Omron Sysmac Studio project Code (Sysmac)_1 (Sysmac Studio 1.64.0.64008, StandardProject)

# Controller new_Controller_0: NX1P2-9B24DT1 version 1.42
Task PrimaryTask (priority 4, period or condition 4000): Program0
Library OEN_Communication_V1_0_22 1.0.22 (contents left out)

TYPE ST_CNC_Cmd : STRUCT  (* CNC DATA *)
    Start : BOOL;  (* CNC Start *)
    Stop : BOOL;  (* CNC Stop *)
    Reset : BOOL;  (* CNC Reset *)
    Busy : BOOL;  (* CNC Busy *)
    FirstPhaseDone : BOOL;  (* CNC Done *)
    LastPhaseDone : BOOL;  (* CNC Done *)
    Progress : INT;  (* CNC Progress *)
    ErrorCode : INT;  (* Erros 1, Error2, Error3 *)
END_STRUCT END_TYPE
TYPE ST_CNC_Timings : STRUCT
    EntryTimeout : BOOL;  (* Flag EntryTimeOut *)
    ProcessTimeout : BOOL;  (* Flag ProcessTimeOut *)
    ExitTimeout : BOOL;  (* Flag ExitEntryTimeOut *)
END_STRUCT END_TYPE

VAR_GLOBAL
    trama : ARRAY[0..4] OF OEN\Modbus\sModbusReq := [(Enable := True, NodeAdr := 1, FunctionCode := Fn15_WriteMultipleCoils, Read := (StartAddressRemote := 0, StartAddressLocal := 0, Count := 0), Write := (StartAddressRemote := 0, StartAddressLocal := 0, Count := 80)), (Enable := True, NodeAdr := 1, FunctionCode := Fn02_ReadDiscreteInputs, Read := (StartAddressRemote := 0, StartAddressLocal := 0, Count := 80), Write := (StartAddressRemote := 0, StartAddressLocal := 0, Count := 0)), (Enable := True, NodeAdr := 1, FunctionCode := Fn04_ReadInputRegisters, Read := (StartAddressRemote := 0, StartAddressLocal := 0, Count := 25), Write := (StartAddressRemote := 0, StartAddressLocal := 0, Count := 0)), (Enable := True, NodeAdr := 1, FunctionCode := Fn16_WriteMultipleRegisters, Read := (StartAddressRemote := 0, StartAddressLocal := 0, Count := 0), Write := (StartAddressRemote := 0, StartAddressLocal := 0, Count := 25)), (Enable := False, NodeAdr := 0, FunctionCode := Fn01_ReadCoils, Read := (StartAddressRemote := 0, StartAddressLocal := 0, Count := 0), Write := (StartAddressRemote := 0, StartAddressLocal := 0, Count := 0))];  (* Trama Responsável pelo invio de informação; published *)
    GB_Cmd : ST_CNC_Cmd;  (* Comandos GreenBases; published *)
    GL_Cmd : ST_CNC_Cmd;  (* Comandos GreenLids *)
    BB_Cmd : ST_CNC_Cmd;  (* Comandos BlueBase *)
    BL_Cmd : ST_CNC_Cmd;  (* Comandos BlueLids *)
    sys_GB_EntrySensor : BOOL;
    sys_GB_ExitSensor AT %W0.01 : BOOL;  (* published *)
    sys_GB_CenterBusy AT %W0.02 : BOOL;  (* published *)
    sys_GB_CenterError AT %W0.03 : BOOL;  (* published *)
END_VAR
VAR_GLOBAL RETAIN
    sys_GB_Progress AT %D0 : INT;  (* published *)
END_VAR
VAR_GLOBAL
    sys_GB_CenterStart AT %W100.00 : BOOL;  (* published *)
    sys_GB_CenterReset AT %W100.01 : BOOL;  (* published *)
    sys_GB_CenterStop AT %W100.02 : BOOL;  (* published *)
    sys_GB_Emitter AT %W100.03 : BOOL;  (* published *)
    sys_GB_EntryConveyor AT %W100.04 : BOOL;  (* published *)
    sys_GB_ExitConveyor AT %W100.05 : BOOL;  (* published *)
    sys_GB_FinalExit_Sensor AT %W100.06 : BOOL;
END_VAR
VAR_GLOBAL RETAIN
    sys_GB_Counter AT %D100 : INT;  (* published *)
END_VAR
VAR_GLOBAL
    sys_GL_EntrySensor AT %W1.00 : BOOL;  (* published *)
    sys_GL_ExitSensor AT %W1.01 : BOOL;  (* published *)
    sys_GL_CenterBusy AT %W1.02 : BOOL;  (* published *)
    sys_GL_CenterError AT %W1.03 : BOOL;  (* published *)
END_VAR
VAR_GLOBAL RETAIN
    sys_GL_Progress AT %D1 : INT;  (* published *)
END_VAR
VAR_GLOBAL
    sys_GL_CenterStart AT %W101.00 : BOOL;  (* published *)
    sys_GL_CenterReset AT %W101.01 : BOOL;  (* published *)
    sys_GL_CenterStop AT %W101.02 : BOOL;  (* published *)
    sys_GL_Emitter AT %W101.03 : BOOL;  (* published *)
    sys_GL_EntryConveyor AT %W101.04 : BOOL;  (* published *)
    sys_GL_ExitConveyor AT %W101.05 : BOOL;  (* published *)
END_VAR
VAR_GLOBAL RETAIN
    sys_GL_Counter AT %D101 : INT;  (* published *)
END_VAR
VAR_GLOBAL
    sys_BB_EntrySensor AT %W2.00 : BOOL;  (* published *)
    sys_BB_ExitSensor AT %W2.01 : BOOL;  (* published *)
    sys_BB_CenterBusy AT %W2.02 : BOOL;  (* published *)
    sys_BB_CenterError AT %W2.03 : BOOL;  (* published *)
END_VAR
VAR_GLOBAL RETAIN
    sys_BB_Progress AT %D2 : INT;  (* published *)
END_VAR
VAR_GLOBAL
    sys_BB_CenterStart AT %W102.00 : BOOL;  (* published *)
    sys_BB_CenterReset AT %W102.01 : BOOL;  (* published *)
    sys_BB_CenterStop AT %W102.02 : BOOL;  (* published *)
    sys_BB_Emitter AT %W102.03 : BOOL;  (* published *)
    sys_BB_EntryConveyor AT %W102.04 : BOOL;  (* published *)
    sys_BB_ExitConveyor AT %W102.05 : BOOL;  (* published *)
END_VAR
VAR_GLOBAL RETAIN
    sys_BB_Counter AT %D102 : INT;  (* published *)
END_VAR
VAR_GLOBAL
    sys_BL_EntrySensor AT %W3.00 : BOOL;  (* published *)
    sys_BL_ExitSensor AT %W3.01 : BOOL;  (* published *)
    sys_BL_CenterBusy AT %W3.02 : BOOL;  (* published *)
    sys_BL_CenterError AT %W3.03 : BOOL;  (* published *)
END_VAR
VAR_GLOBAL RETAIN
    sys_BL_Progress AT %D3 : INT;  (* published *)
END_VAR
VAR_GLOBAL
    sys_BL_CenterStart AT %W103.00 : BOOL;  (* published *)
    sys_BL_CenterReset AT %W103.01 : BOOL;  (* published *)
    sys_BL_CenterStop AT %W103.02 : BOOL;  (* published *)
    sys_BL_Emitter AT %W103.03 : BOOL;  (* published *)
    sys_BL_EntryConveyor AT %W103.04 : BOOL;  (* published *)
    sys_BL_ExitConveyor AT %W103.05 : BOOL;  (* published *)
END_VAR
VAR_GLOBAL RETAIN
    sys_BL_Counter AT %D103 : INT;  (* published *)
END_VAR
VAR_GLOBAL
    sys_StartMain_Button AT %W90.00 : BOOL;  (* published *)
    sys_StopMain_Button AT %W90.01 : BOOL;  (* NC - SafeGuard; published *)
    sys_EmergencyMain_Button AT %W90.02 : BOOL;  (* NC - SafeGuard; published *)
    sys_StackLight_Green AT %W160.00 : BOOL;
    sys_StackLight_Red AT %W160.01 : BOOL;
    sys_StackLight_Yellow AT %W160.02 : BOOL;
    sys_StartLed_Indicator AT %W160.03 : BOOL;
    sys_StopLed_Indicator AT %W160.04 : BOOL;
    sys_EmergencyLed_Indicator AT %W160.05 : BOOL;
END_VAR

PROGRAM Program0
VAR RETAIN
    Master_State : INT := 0;
END_VAR
VAR
    CNC_GB : CNC_Generic;
    CNC_GL : CNC_Generic;
    CNC_BB : CNC_Generic;
    CNC_BL : CNC_Generic;
    TON1_TIME : TIME;  (* Timer_1 *)
    Timer_1 : TON;
END_VAR
VAR_EXTERNAL
    GB_Cmd : ST_CNC_Cmd;
    sys_StartMain_Button : BOOL;
    sys_StopMain_Button : BOOL;
    sys_EmergencyMain_Button : BOOL;
    sys_StackLight_Green : BOOL;
    sys_StackLight_Red : BOOL;
    sys_StartLed_Indicator : BOOL;
    sys_StopLed_Indicator : BOOL;
    sys_GB_EntrySensor : BOOL;
    sys_GB_ExitSensor : BOOL;
    sys_GB_CenterBusy : BOOL;
    sys_GB_CenterError : BOOL;
    sys_GB_Progress : INT;
    sys_GB_CenterStart : BOOL;
    sys_GB_CenterReset : BOOL;
    sys_GB_CenterStop : BOOL;
    sys_GB_Emitter : BOOL;
    sys_GB_EntryConveyor : BOOL;
    sys_GB_ExitConveyor : BOOL;
    sys_GB_Counter : INT;
    sys_GB_FinalExit_Sensor : BOOL;
END_VAR

(* Section Phases_Master: ladder, written here as Structured Text *)

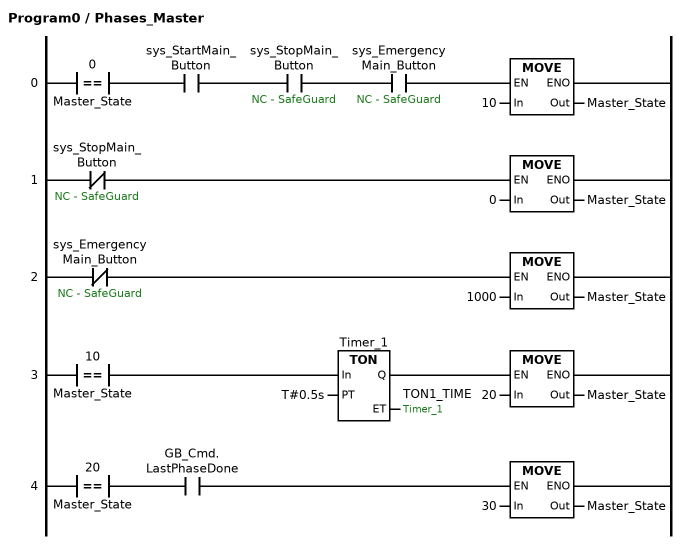
(* Rung 0 *)
IF (0 = Master_State) AND sys_StartMain_Button AND sys_StopMain_Button AND sys_EmergencyMain_Button THEN
    Master_State := 10;
END_IF;
(* Rung 1 *)
IF NOT sys_StopMain_Button THEN Master_State := 0; END_IF;
(* Rung 2 *)
IF NOT sys_EmergencyMain_Button THEN Master_State := 1000; END_IF;
(* Rung 3 *)
Timer_1(In := 10 = Master_State, PT := T#0.5s, ET => TON1_TIME);
IF Timer_1.Q THEN Master_State := 20; END_IF;
(* Rung 4 *)
IF (20 = Master_State) AND GB_Cmd.LastPhaseDone THEN Master_State := 30; END_IF;

(* Section Outputs_Master: ladder, written here as Structured Text *)

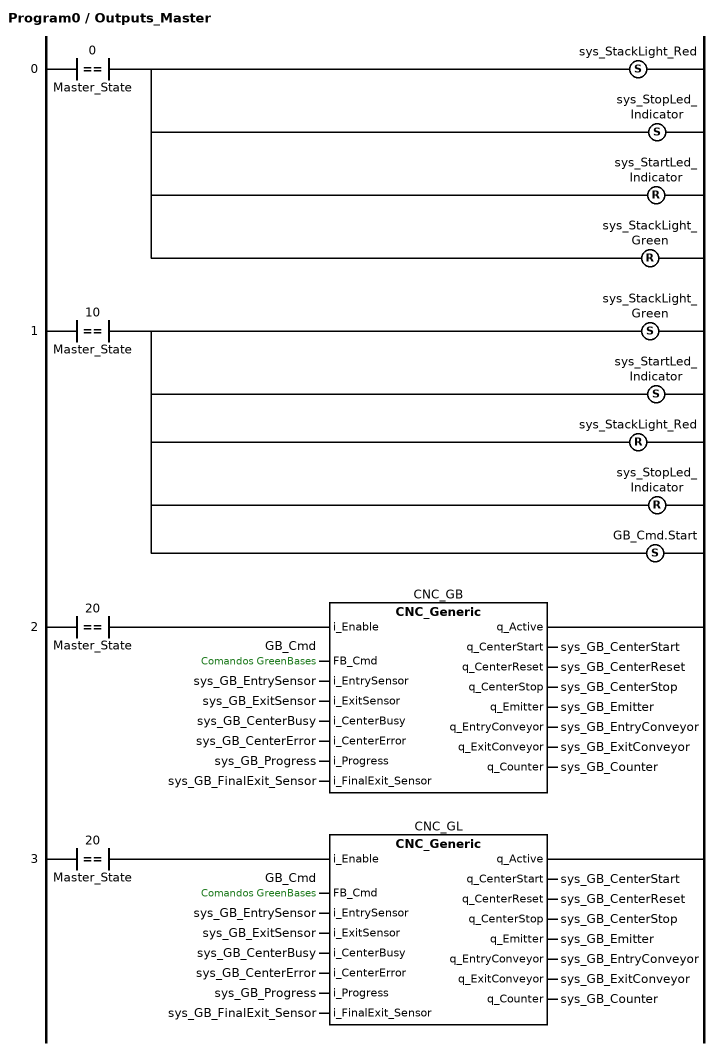
(* Rung 0 *)
IF 0 = Master_State THEN
    sys_StackLight_Red := TRUE;
    sys_StopLed_Indicator := TRUE;
    sys_StartLed_Indicator := FALSE;
    sys_StackLight_Green := FALSE;
END_IF;
(* Rung 1 *)
IF 10 = Master_State THEN
    sys_StackLight_Green := TRUE;
    sys_StartLed_Indicator := TRUE;
    sys_StackLight_Red := FALSE;
    sys_StopLed_Indicator := FALSE;
    GB_Cmd.Start := TRUE;
END_IF;
(* Rung 2 *)
CNC_GB(i_Enable := 20 = Master_State, FB_Cmd := GB_Cmd, i_EntrySensor := sys_GB_EntrySensor, i_ExitSensor := sys_GB_ExitSensor, i_CenterBusy := sys_GB_CenterBusy, i_CenterError := sys_GB_CenterError, i_Progress := sys_GB_Progress, i_FinalExit_Sensor := sys_GB_FinalExit_Sensor, q_CenterStart => sys_GB_CenterStart, q_CenterReset => sys_GB_CenterReset, q_CenterStop => sys_GB_CenterStop, q_Emitter => sys_GB_Emitter, q_EntryConveyor => sys_GB_EntryConveyor, q_ExitConveyor => sys_GB_ExitConveyor, q_Counter => sys_GB_Counter);
(* Rung 3 *)
CNC_GL(i_Enable := 20 = Master_State, FB_Cmd := GB_Cmd, i_EntrySensor := sys_GB_EntrySensor, i_ExitSensor := sys_GB_ExitSensor, i_CenterBusy := sys_GB_CenterBusy, i_CenterError := sys_GB_CenterError, i_Progress := sys_GB_Progress, i_FinalExit_Sensor := sys_GB_FinalExit_Sensor, q_CenterStart => sys_GB_CenterStart, q_CenterReset => sys_GB_CenterReset, q_CenterStop => sys_GB_CenterStop, q_Emitter => sys_GB_Emitter, q_EntryConveyor => sys_GB_EntryConveyor, q_ExitConveyor => sys_GB_ExitConveyor, q_Counter => sys_GB_Counter);
END_PROGRAM

FUNCTION_BLOCK CNC_Generic
VAR
    CNC_State : INT;
    CNC_State_Aux : INT;
    CNC_Timings : ST_CNC_Timings;
    EntryTimer_1 : TON;
    Entry_Timer_1 : TIME;
    Entry_Timer_2 : TIME;
    EntryTimer_2 : TON;
    EntryTimer_3 : TON;
    Entry_Timer_3 : TIME;
    EntryTimer_4 : TON;
    Entry_Timer_4 : TIME;
    EntryTimer_0 : TON;
    Entry_Timer_0 : TIME;
    EntryTimer_5 : TON;
    Entry_Timer_5 : TIME;
    EntryTimer_6 : TON;
    Entry_Timer_6 : TIME;
    EntryTimer_7 : TON;
    Entry_Timer_7 : TIME;
    EntryTimer_8 : TON;
    Entry_Timer_8 : TIME;
END_VAR
VAR_IN_OUT
    FB_Cmd : ST_CNC_Cmd;  (* Busy . *)
END_VAR
VAR_INPUT
    i_Enable : BOOL;
    i_EntrySensor : BOOL;
    i_ExitSensor : BOOL;
    i_CenterBusy : BOOL;
    i_CenterError : BOOL;
    i_Progress : INT;
    i_FinalExit_Sensor : BOOL;
END_VAR
VAR_OUTPUT
    q_Active : BOOL;
    q_CenterStart : BOOL;
    q_CenterReset : BOOL;
    q_CenterStop : BOOL;
    q_Emitter : BOOL;
    q_EntryConveyor : BOOL;
    q_ExitConveyor : BOOL;
    q_Counter : INT;
END_VAR
VAR
    _p1 : BOOL;
    _p2 : BOOL;
    _p3 : BOOL;
    _p4 : BOOL;
END_VAR
(* ladder, written here as Structured Text *)

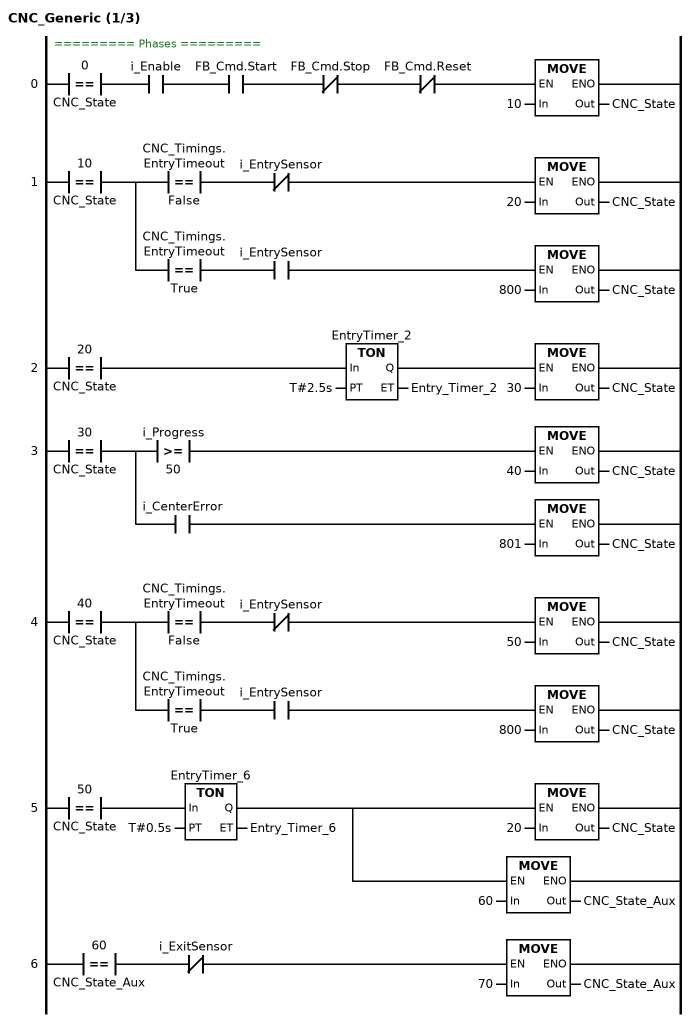
(* Rung 0: ========= Phases ========= *)
IF (0 = CNC_State) AND i_Enable AND FB_Cmd.Start AND NOT FB_Cmd.Stop AND NOT FB_Cmd.Reset THEN
    CNC_State := 10;
END_IF;
(* Rung 1 *)
_p1 := 10 = CNC_State;
IF (10 = CNC_State) AND (CNC_Timings.EntryTimeout = False) AND NOT i_EntrySensor THEN
    CNC_State := 20;
END_IF;
IF _p1 AND (CNC_Timings.EntryTimeout = True) AND i_EntrySensor THEN CNC_State := 800; END_IF;
(* Rung 2 *)
EntryTimer_2(In := 20 = CNC_State, PT := T#2.5s, ET => Entry_Timer_2);
IF EntryTimer_2.Q THEN CNC_State := 30; END_IF;
(* Rung 3 *)
_p2 := 30 = CNC_State;
IF (30 = CNC_State) AND (i_Progress >= 50) THEN CNC_State := 40; END_IF;
IF _p2 AND i_CenterError THEN CNC_State := 801; END_IF;
(* Rung 4 *)
_p3 := 40 = CNC_State;
IF (40 = CNC_State) AND (CNC_Timings.EntryTimeout = False) AND NOT i_EntrySensor THEN
    CNC_State := 50;
END_IF;
IF _p3 AND (CNC_Timings.EntryTimeout = True) AND i_EntrySensor THEN CNC_State := 800; END_IF;
(* Rung 5 *)
EntryTimer_6(In := 50 = CNC_State, PT := T#0.5s, ET => Entry_Timer_6);
IF EntryTimer_6.Q THEN
    CNC_State := 20;
    CNC_State_Aux := 60;
END_IF;
(* Rung 6 *)
IF (60 = CNC_State_Aux) AND NOT i_ExitSensor THEN CNC_State_Aux := 70; END_IF;

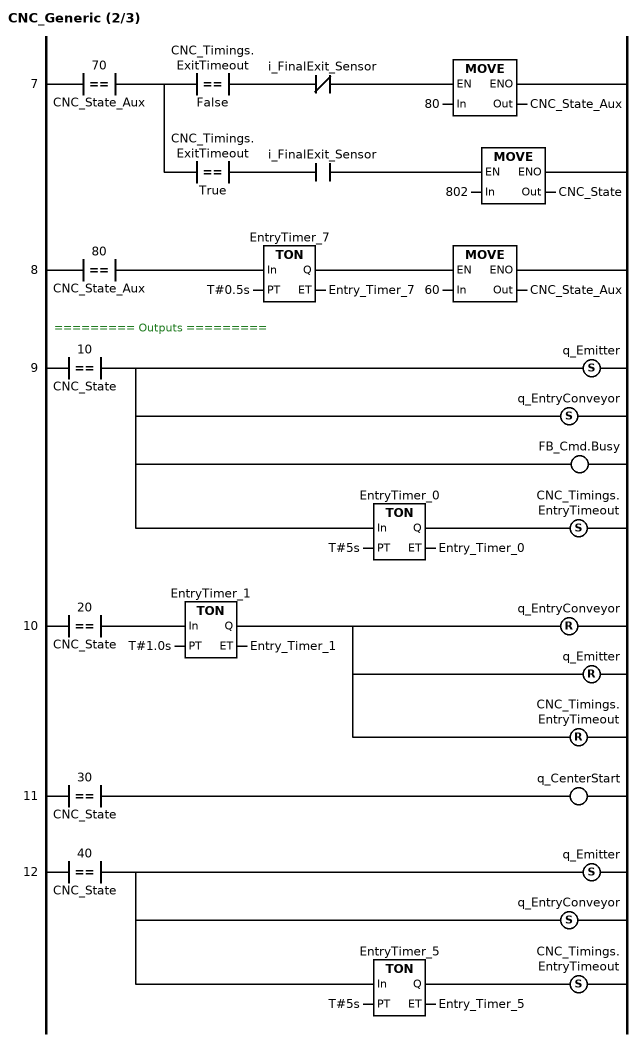
(* Rung 7 *)
_p4 := 70 = CNC_State_Aux;
IF (70 = CNC_State_Aux) AND (CNC_Timings.ExitTimeout = False) AND NOT i_FinalExit_Sensor THEN
    CNC_State_Aux := 80;
END_IF;
IF _p4 AND (CNC_Timings.ExitTimeout = True) AND i_FinalExit_Sensor THEN CNC_State := 802; END_IF;
(* Rung 8 *)
EntryTimer_7(In := 80 = CNC_State_Aux, PT := T#0.5s, ET => Entry_Timer_7);
IF EntryTimer_7.Q THEN CNC_State_Aux := 60; END_IF;
(* Rung 9: ========= Outputs ========= *)
IF 10 = CNC_State THEN
    q_Emitter := TRUE;
    q_EntryConveyor := TRUE;
END_IF;
FB_Cmd.Busy := 10 = CNC_State;
EntryTimer_0(In := 10 = CNC_State, PT := T#5s, ET => Entry_Timer_0);
IF EntryTimer_0.Q THEN CNC_Timings.EntryTimeout := TRUE; END_IF;
(* Rung 10 *)
EntryTimer_1(In := 20 = CNC_State, PT := T#1.0s, ET => Entry_Timer_1);
IF EntryTimer_1.Q THEN
    q_EntryConveyor := FALSE;
    q_Emitter := FALSE;
    CNC_Timings.EntryTimeout := FALSE;
END_IF;
(* Rung 11 *)
q_CenterStart := 30 = CNC_State;
(* Rung 12 *)
IF 40 = CNC_State THEN
    q_Emitter := TRUE;
    q_EntryConveyor := TRUE;
END_IF;
EntryTimer_5(In := 40 = CNC_State, PT := T#5s, ET => Entry_Timer_5);
IF EntryTimer_5.Q THEN CNC_Timings.EntryTimeout := TRUE; END_IF;

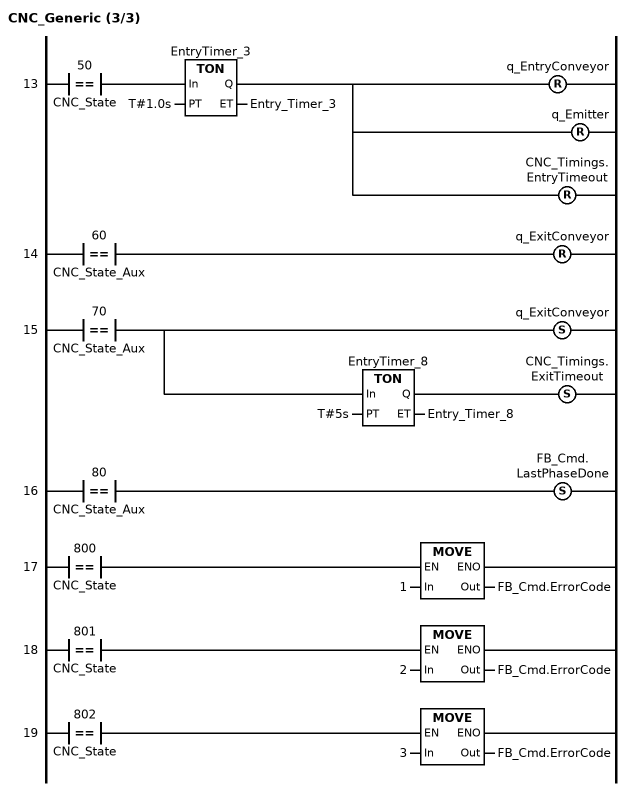
(* Rung 13 *)
EntryTimer_3(In := 50 = CNC_State, PT := T#1.0s, ET => Entry_Timer_3);
IF EntryTimer_3.Q THEN
    q_EntryConveyor := FALSE;
    q_Emitter := FALSE;
    CNC_Timings.EntryTimeout := FALSE;
END_IF;
(* Rung 14 *)
IF 60 = CNC_State_Aux THEN q_ExitConveyor := FALSE; END_IF;
(* Rung 15 *)
IF 70 = CNC_State_Aux THEN q_ExitConveyor := TRUE; END_IF;
EntryTimer_8(In := 70 = CNC_State_Aux, PT := T#5s, ET => Entry_Timer_8);
IF EntryTimer_8.Q THEN CNC_Timings.ExitTimeout := TRUE; END_IF;
(* Rung 16 *)
IF 80 = CNC_State_Aux THEN FB_Cmd.LastPhaseDone := TRUE; END_IF;
(* Rung 17 *)
IF 800 = CNC_State THEN FB_Cmd.ErrorCode := 1; END_IF;
(* Rung 18 *)
IF 801 = CNC_State THEN FB_Cmd.ErrorCode := 2; END_IF;
(* Rung 19 *)
IF 802 = CNC_State THEN FB_Cmd.ErrorCode := 3; END_IF;
END_FUNCTION_BLOCK